Fanuc KAREL source: kx00025.KL

-- PROVISIONAL review KL for V1013-1; original PC SHA256 f1f492bf2b2b2dc3efc9215e9a69d65b5dc62fe7c0c747eb2515d9b2c2964289
-- Incomplete behavior may be omitted. Consult companion uncertainty JSON. Do not deploy.
PROGRAM KX00025
%NOLOCKGROUP
VAR
  I : INTEGER
  J : INTEGER
  B : BOOLEAN
  F : FILE
  S : STRING[80]
-- UNRESOLVED_DECL P type=000102
BEGIN
  -- UNRESOLVED_PC offsets 5-12; opcodes 9D,23
  -- UNRESOLVED_PC offsets 17-21; opcodes 7F
END KX00025
